TYPE ST_MsgBox :
STRUCT
	bShow : BOOL := FALSE;
	sMessageText : STRING(32) := '_just_a_message_';
	sResponse : STRING(32) := '_just_an_response_';
END_STRUCT
END_TYPE

(* stored: Version 1.1.0.1, ProductVersion 3.1.4024.12
   DUT ST_MsgBox: Id {cbeb196d-d592-47b5-b1ed-1e5e17cc6f3f} *)
